// TIA Portal project "sorting task" (V15)

(* hardware
DEVICE "S7300/ET200M station_1"  S7-300 station
   slot 0: "Rail_0"  Rail  6ES7 390-1***0-0AA0
   slot 2: "PLC_1"  CPU 313C-2 DP  6ES7 313-6CF03-0AB0  V2.6
      slot 0: "MPI interface_1"  X1
      slot 1: "DP interface_1"  X2
      slot 2: "DI 16/DO 16_1"  DI16/DO16
      slot 4: "Count_1"  Counter
DEVICE "S7300/ET200M station_2"  S7-300 station
   slot 0: "Rail_0"  Rail  6ES7 390-1***0-0AA0
   slot 2: "PLC_2"  CPU 313C-2 DP  6ES7 313-6CF03-0AB0  V2.6
      slot 0: "MPI interface_1"  X1
      slot 1: "DP interface_1"  X2
      slot 2: "DI 16/DO 16_1"  DI16/DO16
      slot 4: "Count_1"  Counter
*)

// ===== PLC "PLC_1"  CPU 313C-2 DP =====

VAR_GLOBAL   // PLC tag table "Default tag table"
   "Start" AT %I0.5 : Bool;
   "stop" AT %I0.6 : Bool;
   "reset" AT %I0.7 : Bool;
   "L.S" AT %I0.3 : Bool;
   "H.S" AT %I0.4 : Bool;
   "Cyl UP" AT %Q0.0 : Bool;
   "Cyl Down" AT %Q0.1 : Bool;
   "MF" AT %Q0.2 : Bool;
   "MR" AT %Q0.3 : Bool;
   "Suction" AT %Q0.4 : Bool;
   "M1" AT %Q0.5 : Bool;
   "X" AT %M0.0 : Bool;
   "Auto" AT %M41.4 : Bool;
   "Manual" AT %M41.3 : Bool;
   "R1" AT %M0.3 : Bool;
   "R2" AT %M0.4 : Bool;
   "R3" AT %M0.5 : Bool;
   "R4" AT %M0.6 : Bool;
   "R5" AT %M0.7 : Bool;
   "R6" AT %M1.0 : Bool;
   "R7" AT %M1.1 : Bool;
   "R8" AT %M1.2 : Bool;
   "Z1" AT %M2.0 : Bool;
   "Z2" AT %M2.1 : Bool;
   "Z3" AT %M2.2 : Bool;
   "Z4" AT %M2.3 : Bool;
   "Z5" AT %M2.4 : Bool;
   "Z6" AT %M2.5 : Bool;
   "Z7" AT %M2.6 : Bool;
   "Z8" AT %M2.7 : Bool;
   "M11" AT %M32.0 : Bool;
   "M12" AT %M32.1 : Bool;
   "M13" AT %M32.2 : Bool;
   "M14" AT %M32.3 : Bool;
   "M15" AT %M32.4 : Bool;
   "M16" AT %M32.5 : Bool;
   "M17" AT %M32.6 : Bool;
   "M18" AT %M32.7 : Bool;
   "M21" AT %M34.0 : Bool;
   "M22" AT %M34.1 : Bool;
   "M23" AT %M34.2 : Bool;
   "M24" AT %M34.3 : Bool;
   "M25" AT %M34.4 : Bool;
   "M26" AT %M34.5 : Bool;
   "M27" AT %M34.6 : Bool;
   "M28" AT %M34.7 : Bool;
   "P0" AT %M8.0 : Bool;
   "P1" AT %M8.1 : Bool;
   "P2" AT %M8.2 : Bool;
   "P3" AT %M8.3 : Bool;
   "P4" AT %M8.4 : Bool;
   "P5" AT %M8.5 : Bool;
   "P6" AT %M8.6 : Bool;
   "P7" AT %M8.7 : Bool;
   "N0" AT %M9.0 : Bool;
   "N1" AT %M9.1 : Bool;
   "N2" AT %M9.2 : Bool;
   "N3" AT %M9.3 : Bool;
   "N4" AT %M9.4 : Bool;
   "N5" AT %M9.5 : Bool;
   "N6" AT %M9.6 : Bool;
   "N7" AT %M9.7 : Bool;
   "MW20" AT %MW20 : Word;
   "MD100" AT %MD100 : DInt;
   "MD104" AT %MD104 : DInt;
   "C0" AT %M10.0 : Bool;
   "C1" AT %M10.1 : Bool;
   "C2" AT %M10.2 : Bool;
   "C3" AT %M10.3 : Bool;
   "C4" AT %M10.4 : Bool;
   "C5" AT %M10.5 : Bool;
   "C6" AT %M10.6 : Bool;
   "C7" AT %M10.7 : Bool;
   "TON0" AT %M11.0 : Timer;
   "TON1" AT %M11.1 : Bool;
   "TON2" AT %M11.2 : Bool;
   "TON3" AT %M11.3 : Bool;
   "TON4" AT %M11.4 : Bool;
   "TON5" AT %M11.5 : Bool;
   "TON6" AT %M11.6 : Bool;
   "TON7" AT %M11.7 : Bool;
   "T1" AT %M12.0 : Bool;
   "T2" AT %M12.1 : Bool;
   "T3" AT %M12.2 : Bool;
   "T4" AT %M12.3 : Bool;
   "T5" AT %M12.4 : Bool;
   "T6" AT %M12.5 : Bool;
   "T7" AT %M12.6 : Bool;
   "T0" AT %M12.7 : Bool;
   "Large" AT %M13.0 : Bool;
   "small" AT %M13.1 : Bool;
   "B" AT %M13.2 : Bool;
   "u0" AT %M13.3 : Bool;
   "u1" AT %M13.4 : Bool;
   "u2" AT %M13.5 : Bool;
   "u3" AT %M13.6 : Bool;
   "u4" AT %M13.7 : Bool;
   "u5" AT %M14.0 : Bool;
   "u6" AT %M14.1 : Bool;
   "u7" AT %M14.2 : Bool;
   "u8" AT %M14.3 : Bool;
   "u9" AT %M14.4 : Bool;
   "u10" AT %M14.5 : Bool;
   "u11" AT %M14.6 : Bool;
   "u12" AT %M14.7 : Bool;
   "mw88" AT %MW88 : Word;
   "MW30" AT %MW30 : Word;
   "MW32" AT %MW32 : Word;
   "MW34" AT %MW34 : Word;
   "Y" AT %M4.0 : Bool;
   "Y1" AT %M4.1 : Bool;
   "Y2" AT %M4.2 : Bool;
   "Y3" AT %M4.3 : Bool;
   "smll" AT %M4.4 : Bool;
   "up" AT %M40.0 : Bool;
   "down" AT %M40.1 : Bool;
   "left" AT %M40.2 : Bool;
   "right" AT %M40.3 : Bool;
   "suc" AT %M40.4 : Bool;
   "forword" AT %M40.5 : Bool;
   "qw50" AT %QW50 : Word;
   "qw52" AT %QW52 : Word;
   "qw54" AT %QW54 : Word;
   "iw50" AT %IW50 : Word;
   "iw52" AT %IW52 : Word;
   "iw0" AT %IW0 : Word;
   "mw40" AT %MW40 : Word;
   "qw0" AT %QW0 : Word;
   "staart" AT %M41.0 : Bool;
   "stoop" AT %M41.1 : Bool;
   "rese" AT %M41.2 : Bool;
END_VAR

DATA_BLOCK "0"   // DB1
{ S7_Optimized_Access := 'FALSE' }
VERSION : 0.1
// stored: InstanceOfName Negative Age
"Negative Age"
BEGIN
END_DATA_BLOCK

DATA_BLOCK "2"   // DB2
{ S7_Optimized_Access := 'FALSE' }
VERSION : 0.1
// stored: InstanceOfName Negative Age
"Negative Age"
BEGIN
END_DATA_BLOCK

DATA_BLOCK "3"   // DB3
{ S7_Optimized_Access := 'FALSE' }
VERSION : 0.1
// stored: InstanceOfName positive age
"positive age"
BEGIN
END_DATA_BLOCK

DATA_BLOCK "6"   // DB4
{ S7_Optimized_Access := 'FALSE' }
VERSION : 0.1
// stored: InstanceOfName Negative Age
"Negative Age"
BEGIN
END_DATA_BLOCK

DATA_BLOCK "4"   // DB5
{ S7_Optimized_Access := 'FALSE' }
VERSION : 0.1
// stored: InstanceOfName Negative Age
"Negative Age"
BEGIN
END_DATA_BLOCK

DATA_BLOCK "5"   // DB6
{ S7_Optimized_Access := 'FALSE' }
VERSION : 0.1
// stored: InstanceOfName positive age
"positive age"
BEGIN
END_DATA_BLOCK

DATA_BLOCK "7"   // DB7
{ S7_Optimized_Access := 'FALSE' }
VERSION : 0.1
// stored: InstanceOfName positive age
"positive age"
BEGIN
END_DATA_BLOCK

DATA_BLOCK "fb small r8"   // DB8
{ S7_Optimized_Access := 'FALSE' }
VERSION : 0.1
// stored: InstanceOfName FB.SMALL
"FB.SMALL"
BEGIN
END_DATA_BLOCK

DATA_BLOCK "FB.LARGE_R1"   // DB9
{ S7_Optimized_Access := 'FALSE' }
VERSION : 0.1
// stored: InstanceOfName FB.LARGE
"FB.LARGE"
BEGIN
END_DATA_BLOCK

DATA_BLOCK "FB.SMALL_r7"   // DB10
{ S7_Optimized_Access := 'FALSE' }
VERSION : 0.1
// stored: InstanceOfName FB.SMALL
"FB.SMALL"
BEGIN
END_DATA_BLOCK

DATA_BLOCK "FB.SMALL_R6"   // DB11
{ S7_Optimized_Access := 'FALSE' }
VERSION : 0.1
// stored: InstanceOfName FB.SMALL
"FB.SMALL"
BEGIN
END_DATA_BLOCK

DATA_BLOCK "FB.SMALL_R5"   // DB12
{ S7_Optimized_Access := 'FALSE' }
VERSION : 0.1
// stored: InstanceOfName FB.SMALL
"FB.SMALL"
BEGIN
END_DATA_BLOCK

DATA_BLOCK "FB.SMALL_R4"   // DB13
{ S7_Optimized_Access := 'FALSE' }
VERSION : 0.1
// stored: InstanceOfName FB.SMALL
"FB.SMALL"
BEGIN
END_DATA_BLOCK

DATA_BLOCK "FB.SMALL_R3"   // DB14
{ S7_Optimized_Access := 'FALSE' }
VERSION : 0.1
// stored: InstanceOfName FB.SMALL
"FB.SMALL"
BEGIN
END_DATA_BLOCK

DATA_BLOCK "FB.SMALL_R2"   // DB15
{ S7_Optimized_Access := 'FALSE' }
VERSION : 0.1
// stored: InstanceOfName FB.SMALL
"FB.SMALL"
BEGIN
END_DATA_BLOCK

DATA_BLOCK "FB.SMALL_R1"   // DB16
{ S7_Optimized_Access := 'FALSE' }
VERSION : 0.1
// stored: InstanceOfName FB.SMALL
"FB.SMALL"
BEGIN
END_DATA_BLOCK

DATA_BLOCK "FB.LARGE_R2"   // DB17
{ S7_Optimized_Access := 'FALSE' }
VERSION : 0.1
// stored: InstanceOfName FB.LARGE
"FB.LARGE"
BEGIN
END_DATA_BLOCK

DATA_BLOCK "FB.LARGE_R3"   // DB18
{ S7_Optimized_Access := 'FALSE' }
VERSION : 0.1
// stored: InstanceOfName FB.LARGE
"FB.LARGE"
BEGIN
END_DATA_BLOCK

DATA_BLOCK "FB.LARGE_R4"   // DB19
{ S7_Optimized_Access := 'FALSE' }
VERSION : 0.1
// stored: InstanceOfName FB.LARGE
"FB.LARGE"
BEGIN
END_DATA_BLOCK

DATA_BLOCK "FB.LARGE_R5"   // DB20
{ S7_Optimized_Access := 'FALSE' }
VERSION : 0.1
// stored: InstanceOfName FB.LARGE
"FB.LARGE"
BEGIN
END_DATA_BLOCK

DATA_BLOCK "FB.LARGE_R6"   // DB21
{ S7_Optimized_Access := 'FALSE' }
VERSION : 0.1
// stored: InstanceOfName FB.LARGE
"FB.LARGE"
BEGIN
END_DATA_BLOCK

DATA_BLOCK "FB.LARGE_R7"   // DB22
{ S7_Optimized_Access := 'FALSE' }
VERSION : 0.1
// stored: InstanceOfName FB.LARGE
"FB.LARGE"
BEGIN
END_DATA_BLOCK

DATA_BLOCK "FB.LARGE_R8"   // DB23
{ S7_Optimized_Access := 'FALSE' }
VERSION : 0.1
// stored: InstanceOfName FB.LARGE
"FB.LARGE"
BEGIN
END_DATA_BLOCK

DATA_BLOCK "FB.R1"   // DB24
{ S7_Optimized_Access := 'FALSE' }
VERSION : 0.1
// stored: InstanceOfName FB.MR
"FB.MR"
BEGIN
END_DATA_BLOCK

DATA_BLOCK "FB.R2"   // DB25
{ S7_Optimized_Access := 'FALSE' }
VERSION : 0.1
// stored: InstanceOfName FB.MR
"FB.MR"
BEGIN
END_DATA_BLOCK

DATA_BLOCK "FB.R3"   // DB26
{ S7_Optimized_Access := 'FALSE' }
VERSION : 0.1
// stored: InstanceOfName FB.MR
"FB.MR"
BEGIN
END_DATA_BLOCK

DATA_BLOCK "FB.R4"   // DB27
{ S7_Optimized_Access := 'FALSE' }
VERSION : 0.1
// stored: InstanceOfName FB.MR
"FB.MR"
BEGIN
END_DATA_BLOCK

DATA_BLOCK "FB.R5"   // DB28
{ S7_Optimized_Access := 'FALSE' }
VERSION : 0.1
// stored: InstanceOfName FB,MF
"FB,MF"
BEGIN
END_DATA_BLOCK

DATA_BLOCK "FB.R6"   // DB29
{ S7_Optimized_Access := 'FALSE' }
VERSION : 0.1
// stored: InstanceOfName FB,MF
"FB,MF"
BEGIN
END_DATA_BLOCK

DATA_BLOCK "FB.R7"   // DB30
{ S7_Optimized_Access := 'FALSE' }
VERSION : 0.1
// stored: InstanceOfName FB,MF
"FB,MF"
BEGIN
END_DATA_BLOCK

DATA_BLOCK "FB.R8"   // DB31
{ S7_Optimized_Access := 'FALSE' }
VERSION : 0.1
// stored: InstanceOfName FB,MF
"FB,MF"
BEGIN
END_DATA_BLOCK

DATA_BLOCK "Negative Age_last"   // DB33
{ S7_Optimized_Access := 'FALSE' }
VERSION : 0.1
// stored: InstanceOfName Negative Age
"Negative Age"
BEGIN
END_DATA_BLOCK

FUNCTION_BLOCK "Negative Age"   // FB1, SCL
{ S7_Optimized_Access := 'FALSE' }
VERSION : 0.1
   VAR_INPUT
      in : Bool;
   END_VAR
   VAR_OUTPUT
      out : Bool;
   END_VAR
   VAR_IN_OUT
      y : Bool;
   END_VAR
BEGIN
   #out := NOT #in AND #y;
   #y := #y;
END_FUNCTION_BLOCK

FUNCTION_BLOCK "positive age"   // FB2, SCL
{ S7_Optimized_Access := 'FALSE' }
VERSION : 0.1
   VAR_INPUT
      in : Bool;
   END_VAR
   VAR_OUTPUT
      out : Bool;
   END_VAR
   VAR_IN_OUT
      y : Bool;
   END_VAR
BEGIN
   #out := #in AND NOT #y;
   #y := #in;
END_FUNCTION_BLOCK

FUNCTION_BLOCK "Block_1"   // FB3, LAD
{ S7_Optimized_Access := 'FALSE' }
VERSION : 0.1
   VAR_TEMP   // added for the SCL form of the ladder/FBD networks
      _s5time1 : S5Time;
   END_VAR
BEGIN

REGION Network 1
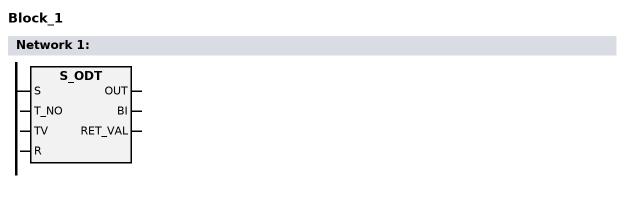
   RUNG wire#powerrail
      S_ODT(T_NO :=, TV :=, R :=, BI =>, RET_VAL =>)
   END_RUNG
   // the same network as SCL:
   #_s5time1 := S_ODT(S := TRUE);
END_REGION
END_FUNCTION_BLOCK

FUNCTION_BLOCK "FB.SMALL"   // FB4, SCL
{ S7_Optimized_Access := 'FALSE' }
VERSION : 0.1
BEGIN
   "R8" := NOT "M18";
   "R7" := NOT "M17" AND NOT "R8";
   "R6" := NOT "M16" AND NOT "R8" AND NOT "R7" ;
   "R5" := NOT "M15" AND NOT "R8" AND NOT "R7" AND NOT "R6" ;
   "R4" := NOT "M14" AND NOT "R8" AND NOT "R7" AND NOT "R6" AND NOT "R5";
   "R3" := NOT "M13" AND NOT "R8" AND NOT "R7" AND NOT "R6" AND NOT "R5" AND NOT "R4" ;
   "R2" := NOT "M12" AND NOT "R8" AND NOT "R7" AND NOT "R6" AND NOT "R5" AND NOT "R4" AND NOT "R3";
   "R1" := NOT "M11" AND NOT "R8" AND NOT "R7" AND NOT "R6" AND NOT "R5" AND NOT "R4" AND NOT "R3" AND NOT "R2";
   IF "R8"=1 AND "Y"=1 THEN
       SET(S_BIT:="M18",N:=1);
   END_IF;
   IF "R7" = 1 AND "Y" = 1 THEN
       SET(S_BIT := "M17",N := 2);
   END_IF;
   IF "R6" = 1 AND "Y" = 1 THEN
       SET(S_BIT := "M16",N := 3);
   END_IF;
   IF "R5" = 1 AND "Y" = 1 THEN
       SET(S_BIT := "M15",N := 4);
   END_IF;
   IF "R4" = 1 AND "Y" = 1 THEN
       SET(S_BIT := "M14",N := 5);
   END_IF;
   IF "R3" = 1 AND "Y" = 1 THEN
       SET(S_BIT := "M13", N := 6);
   END_IF;
   IF "R2" = 1 AND "Y" = 1 THEN
       SET(S_BIT := "M12", N := 7);
   END_IF;
   IF "R1" = 1 AND "Y" = 1 THEN
       SET(S_BIT := "M11", N := 8);
   END_IF;
END_FUNCTION_BLOCK

FUNCTION_BLOCK "FB.LARGE"   // FB5, SCL
{ S7_Optimized_Access := 'FALSE' }
VERSION : 0.1
BEGIN
   "R1" := "M21";
   "R2" := "M22" AND NOT "R1";
   "R3" := "M23" AND NOT "R1" AND NOT "R2";
   "R4" := "M24" AND NOT "R1" AND NOT "R2" AND NOT "R3";
   "R5" := "M25" AND NOT "R1" AND NOT "R2" AND NOT "R3" AND NOT "R4";
   "R6" := "M26" AND NOT "R1" AND NOT "R2" AND NOT "R3" AND NOT "R4" AND NOT "R5";
   "R7" := "M27" AND NOT "R1" AND NOT "R2" AND NOT "R3" AND NOT "R4" AND NOT "R5" AND NOT "R6";
   "R8" := "M28" AND NOT "R1" AND NOT "R2" AND NOT "R3" AND NOT "R4" AND NOT "R5" AND NOT "R6" AND NOT "R7";
   IF "R1"=1 AND "Y"=1THEN
       RESET(S_BIT:="M21", N:=1);
   END_IF;
   IF "R2" = 1 AND "Y" = 1 THEN
       RESET(S_BIT := "M22",
             N := 2);
   END_IF;
   IF "R3" = 1 AND "Y" = 1 THEN
       RESET(S_BIT := "M23",
             N := 3);
   END_IF;
   IF "R4" = 1 AND "Y" = 1 THEN
       RESET(S_BIT := "M24",
             N := 4);
   END_IF;
   IF "R5" = 1 AND "Y" = 1 THEN
       RESET(S_BIT := "M25",
             N := 5);
   END_IF;
   IF "R6" = 1 AND "Y" = 1 THEN
       RESET(S_BIT := "M26",
             N := 6);
   END_IF;
   IF "R7" = 1 AND "Y" = 1 THEN
       RESET(S_BIT := "M27",
             N := 7);
   END_IF;
   IF "R8" = 1 AND "Y" = 1 THEN
       RESET(S_BIT := "M28",
             N := 8);
   END_IF;
END_FUNCTION_BLOCK

FUNCTION_BLOCK "FB.MR"   // FB6, SCL
{ S7_Optimized_Access := 'FALSE' }
VERSION : 0.1
   VAR_INPUT
      MD110 : DInt;
   END_VAR
   VAR
      P00 : Bool;
      T00 : Bool;
      T11 : Bool;
      T22 : Bool;
      T33 : Bool;
      T44 : Bool;
      T55 : Bool;
      T66 : Bool;
      T77 : Bool;
      T88 : Bool;
      MW88 : Word;
      U00 : Bool;
      U11 : Bool;
      U22 : Bool;
      U33 : Bool;
   END_VAR
BEGIN
   "7"(in:="T1",out=>#P00, y:=#U00);
   IF #P00=1 THEN
       SET(S_BIT:="Cyl Down",  N:=9);
   END_IF;

   #MW88:= S_ODT(T_NO:=10, S:="Cyl Down"AND NOT "Suction", TV:=S5T#500MS, Q=>#T11);
   IF #T11=1 THEN
       RESET(S_BIT:="Cyl Down",
             N:=10);
       SET(S_BIT:="Suction",
           N:=11);
       SET(S_BIT:="Cyl UP",
           N:=12);
   END_IF;

   #MW88 := S_ODT(T_NO := 11, S := "Cyl UP" AND "Suction", TV := S5T#500MS, Q => #T22);
   IF #T22 = 1 THEN
       RESET(S_BIT := "Cyl UP",
             N := 13);
       SET(S_BIT := "MR",
           N := 14);
       SET(S_BIT := "Y",
           N := 15);
   END_IF;
   IF "MD100" < #MD110 AND "Suction" = 1 THEN
       RESET(S_BIT := "MR",
             N := 16);
   END_IF;
   IF "R1" = 1 AND "Suction" = 1 AND "MR" = 0 THEN
       SET(S_BIT := "Cyl Down",
           N := 17);
   END_IF;
   #MW88 := S_ODT(T_NO := 12, S := "Cyl Down" AND "Suction", TV := S5T#500MS, Q => #T33);
   IF #T33 = 1 THEN
       RESET(S_BIT := "Cyl Down",
             N := 18);
       RESET(S_BIT := "Suction",
             N := 19);
       SET(S_BIT := "Cyl UP",
           N := 20);
   END_IF;
   #MW88 := S_ODT(T_NO := 13, S := "Cyl UP" AND NOT "Suction", TV := S5T#500MS, Q => #T44);
   IF #T44 = 1 THEN
       RESET(S_BIT := "Cyl UP",
             N := 21);
       RESET(S_BIT := "Y",
             N := 22);
   END_IF;
END_FUNCTION_BLOCK

FUNCTION_BLOCK "FB,MF"   // FB7, SCL
{ S7_Optimized_Access := 'FALSE' }
VERSION : 0.1
   VAR_INPUT
      MD110 : DInt;
   END_VAR
   VAR
      P00 : Bool;
      T00 : Bool;
      T11 : Bool;
      T22 : Bool;
      T33 : Bool;
      T44 : Bool;
      T55 : Bool;
      T66 : Bool;
      T77 : Bool;
      T88 : Bool;
      MW88 : Word;
      U00 : Bool;
      U11 : Bool;
      U22 : Bool;
      U33 : Bool;
   END_VAR
BEGIN
   "7"(in := "T1",
       out => #P00,
       y := #U00);
   IF #P00 = 1 THEN
       SET(S_BIT := "Cyl Down",
           N := 9);
   END_IF;

   #MW88 := S_ODT(T_NO := 10, S := "Cyl Down" AND NOT "Suction", TV := S5T#500MS, Q => #T11);
   IF #T11 = 1 THEN
       RESET(S_BIT := "Cyl Down",
             N := 10);
       SET(S_BIT := "Suction",
           N := 11);
       SET(S_BIT := "Cyl UP",
           N := 12);
   END_IF;

   #MW88 := S_ODT(T_NO := 11, S := "Cyl UP" AND "Suction", TV := S5T#500MS, Q => #T22);
   IF #T22 = 1 THEN
       RESET(S_BIT := "Cyl UP",
             N := 13);
       SET(S_BIT := "MF",
           N := 14);
       SET(S_BIT := "Y",
           N := 15);
   END_IF;
   IF "MD100" > #MD110 AND "Suction" = 1 THEN
       RESET(S_BIT := "MF",
             N := 16);
   END_IF;
   IF "R1" = 1 AND "Suction" = 1 AND "MR" = 0 THEN
       SET(S_BIT := "Cyl Down",
           N := 17);
   END_IF;
   #MW88 := S_ODT(T_NO := 12, S := "Cyl Down" AND "Suction", TV := S5T#500MS, Q => #T33);
   IF #T33 = 1 THEN
       RESET(S_BIT := "Cyl Down",
             N := 18);
       RESET(S_BIT := "Suction",
             N := 19);
       SET(S_BIT := "Cyl UP",
           N := 20);
   END_IF;
   #MW88 := S_ODT(T_NO := 13, S := "Cyl UP" AND NOT "Suction", TV := S5T#500MS, Q => #T44);
   IF #T44 = 1 THEN
       RESET(S_BIT := "Cyl UP",
             N := 21);
       RESET(S_BIT:="Y",
             N:=22);

   END_IF;
END_FUNCTION_BLOCK

ORGANIZATION_BLOCK "Main"   // OB1, SCL
TITLE = "Main Program Sweep (Cycle)"
{ S7_Optimized_Access := 'FALSE' }
VERSION : 0.1
   VAR_TEMP
      OB1_EV_CLASS : Byte;   // Bits 0-3 = 1 (Coming event), Bits 4-7 = 1 (Event class 1)
      OB1_SCAN_1 : Byte;   // 1 (Cold restart scan 1 of OB 1), 3 (Scan 2-n of OB 1)
      OB1_PRIORITY : Byte;   // Priority of OB Execution
      OB1_OB_NUMBR : Byte;   // 1 (Organization block 1, OB1)
      OB1_RESERVED_1 : Byte;   // Reserved for system
      OB1_RESERVED_2 : Byte;   // Reserved for system
      OB1_PREV_CYCLE : Int;   // Cycle time of previous OB1 scan (milliseconds)
      OB1_MIN_CYCLE : Int;   // Minimum cycle time of OB1 (milliseconds)
      OB1_MAX_CYCLE : Int;   // Maximum cycle time of OB1 (milliseconds)
      OB1_DATE_TIME : Date_And_Time;   // Date and time OB1 started
   END_VAR
BEGIN
   REGION "X"
       "X" := ("Start" OR "X" OR "staart") AND "stop" AND "stoop" AND "Auto";
       "5"(in:="X",out=>"P1", y:="u4");
       IF "P1"=1 AND "X"=1  THEN
           "MW32" := "MW30";
           "MW34" := "MW30";
           SET(S_BIT:= "Y1",
               N:=50);

       END_IF;


   END_REGION

   REGION encoder
       "encoder"(LADDR:=16#300,
                 CHANNEL:=0,
                 SW_GATE:="Y1",
                 COUNTVAL=>"MD100");

              END_REGION


   IF "MD100"<5 AND "MD100">-5 THEN
       "M1":="X" AND NOT "Suction";
   ELSE
       "M1" := 0;
   END_IF;

   "0"(in:="H.S", out=>"Large", y:="N0");
   "2"(in:="L.S",out=>"N1", y:="u0");
   "small" := "N1" AND NOT "H.S" AND NOT "Large";

   IF "MD100"<5 AND "MD100">-5 THEN
       "3"(in:=TRUE, out=>"P0", y:="u1");
       IF "MD100"<5 AND "MD100">-5 AND "P0"=1 THEN
           RESET(S_BIT:="Large",
                 N:=32);
           RESET(S_BIT:="small",
                 N:=33);
           RESET(S_BIT:="smll",
                 N:=34);
           RESET(S_BIT := "B",
                 N := 35);
       END_IF;
   END_IF;

   "6"(in:="L.S",out=>"N2", y:="u2");
   "mw88" := S_CU(C_NO := 106, CU := "N2", R:="u8", CV=>"MW20");

   REGION RePosition
       "4"(in := "Suction",
      out => "N3",
      y := "u3");
       IF "N3" = 1 THEN
           SET(S_BIT := "B",
          N := 40);
       END_IF;
       "mw88" := S_ODT(T_NO := 1, S := "B", TV := s5t#600ms, Q => "T2");
       (*
       لو فيه مشكله ان الماتور لما ييجي يرجع للنص 
       ومش بيقف ساعتها اعمل ايلسي لل الكود اللي جاي
       *)
       IF "MD100" < -5 AND "T2" = 1 THEN
           "MF" := 1;

       END_IF;
       IF "MD100" > 5 AND "T2" = 1 THEN
           "MR" := 1;
       END_IF;
   END_REGION


   (*
   التايمر اللي تحت ده الوقت بتاعه هبتغير علي حسب الوقت اللي هيقف فيه السير
   *)
   IF "N1" = 1 THEN
       SET(S_BIT := "smll",
           N := 31);
   END_IF;


   "mw88" := S_ODT(T_NO := 3, S := "smll", TV := S5T#1.5S, Q=>"T1");
   IF "T1" = 1 THEN
       RESET(S_BIT := "M1",
             N := 30);
   END_IF;

   REGION small

   IF "T1" = 1 AND "small" = 1 AND "MW20" = 1 THEN
       "fb small r8"();
   END_IF;
   IF "T1" = 1 AND "small" = 1 AND "MW20" = 2 THEN
       "FB.SMALL_r7"();
   END_IF;
   IF "T1" = 1 AND "small" = 1 AND "MW20" = 3 THEN
       "FB.SMALL_R6"();
   END_IF;
   IF "T1" = 1 AND "small" = 1 AND "MW20" = 4 THEN
       "FB.SMALL_R5"();
   END_IF;
   IF "T1" = 1 AND "small" = 1 AND "MW20" = 5 THEN
       "FB.SMALL_R4"();
   END_IF;
   IF "T1" = 1 AND "small" = 1 AND "MW20" = 6 THEN
       "FB.SMALL_R3"();
   END_IF;
   IF "T1" = 1 AND "small" = 1 AND "MW20" = 7 THEN
       "FB.SMALL_R2"();
   END_IF;
   IF "T1" = 1 AND "small" = 1 AND "MW20" = 8 THEN
       "FB.SMALL_R1"();
   END_IF;

   END_REGION

   REGION large
       IF "Large" = 1 AND "T1" = 1 AND "MW20" = 1 THEN
           "FB.LARGE_R1"();
       END_IF;
       IF "Large" = 1 AND "T1" = 1 AND "MW20" = 2 THEN
           "FB.LARGE_R2"();
       END_IF;
       IF "Large" = 1 AND "T1" = 1 AND "MW20" = 2 THEN
           "FB.LARGE_R3"();
       END_IF;
       IF "Large" = 1 AND "T1" = 1 AND "MW20" = 2 THEN
           "FB.LARGE_R4"();
       END_IF;
       IF "Large" = 1 AND "T1" = 1 AND "MW20" = 2 THEN
           "FB.LARGE_R5"();
       END_IF;
       IF "Large" = 1 AND "T1" = 1 AND "MW20" = 2 THEN
           "FB.LARGE_R6"();
       END_IF;
       IF "Large" = 1 AND "T1" = 1 AND "MW20" = 2 THEN
           "FB.LARGE_R7"();
       END_IF;
       IF "Large" = 1 AND "T1" = 1 AND "MW20" = 2 THEN
           "FB.LARGE_R8"();
       END_IF;

   END_REGION

   REGION POSITION R1
       IF "R1" = 1 THEN
           "FB.R1"(-500);
       END_IF;
   END_REGION

   REGION POSITION R2
       IF "R2" = 1 THEN
           "FB.R2"(-400);
       END_IF;
   END_REGION

   REGION POSITION R3
       IF "R3" = 1 THEN
           "FB.R3"(-300);
       END_IF;
   END_REGION

   REGION POSITION R4
       IF "R4" = 1 THEN
           "FB.R4"(-200);
       END_IF;
   END_REGION

   REGION POSITION R5
       IF "R5" = 1 THEN
           "FB.R5"(200);
       END_IF;
   END_REGION

   REGION POSITION R6
       IF "R6" =1 THEN
      "FB.R6"(300);
       END_IF;
   END_REGION

   REGION POSITION R7
       IF "R7" = 1 THEN
           "FB.R7"(400);
       END_IF;
   END_REGION

   REGION POSITION R8
       IF "R8" = 1 THEN
           "FB.R8"(500);
       END_IF;
   END_REGION

   REGION close program
       "Negative Age_last"(in:="B", out=>"N5",y:="u7");
       IF "N5" = 1 AND "MW20" = 8 THEN
           RESET(S_BIT:="X",
                 N:=41);
           "u8" := 1;

       END_IF;

   END_REGION

   REGION reset
       IF "reset" = 1 OR "rese"=1 THEN
           SET(S_BIT := "Y2",
               N := 51);
       END_IF;
       IF "Y2" = 1 THEN
           IF "MD100" > 5 THEN
               "MR" := 1;
           ELSE
               "MR" := 0;
           END_IF;
           IF "MD100" < -5 THEN
               "MF" := 1;
           ELSE
               "MF" := 0;
           END_IF;
           IF "MD100"<10 AND "MD100">-10 THEN
               RESET(S_BIT := "Y2",
                     N := 45);
           END_IF;

       END_IF;
   END_REGION

   REGION manual
       IF "Manual"=1 AND "Auto" =0 THEN
           "Cyl Down" := "down";
           "Cyl UP" := "up";
           "MF" := "left";
           "MR" := "right";
           "Suction" := "suc";
           "M1" := "forword";
       END_IF;

   END_REGION

   REGION communication
       "qw50" := "iw0";
       "qw52" := "qw0"; 
       "mw40" := "iw50";
       "MW30" := "iw52";
       "qw54" := "MW30";



   END_REGION
END_ORGANIZATION_BLOCK

// ===== PLC "PLC_2"  CPU 313C-2 DP =====

VAR_GLOBAL   // PLC tag table "Default tag table"
   "mw0" AT %MW0 : Word;
   "iw50" AT %IW50 : Word;
   "iw52" AT %IW52 : Word;
   "iw54" AT %IW54 : Word;
   "qw50" AT %QW50 : Word;
   "qw52" AT %QW52 : Word;
   "mw10" AT %QW54 : Word;
   "mw40" AT %QW56 : Word;
   "mw30" AT %QW58 : Word;
END_VAR

ORGANIZATION_BLOCK "Main"   // OB1, SCL
TITLE = "Main Program Sweep (Cycle)"
{ S7_Optimized_Access := 'FALSE' }
VERSION : 0.1
   VAR_TEMP
      OB1_EV_CLASS : Byte;   // Bits 0-3 = 1 (Coming event), Bits 4-7 = 1 (Event class 1)
      OB1_SCAN_1 : Byte;   // 1 (Cold restart scan 1 of OB 1), 3 (Scan 2-n of OB 1)
      OB1_PRIORITY : Byte;   // Priority of OB Execution
      OB1_OB_NUMBR : Byte;   // 1 (Organization block 1, OB1)
      OB1_RESERVED_1 : Byte;   // Reserved for system
      OB1_RESERVED_2 : Byte;   // Reserved for system
      OB1_PREV_CYCLE : Int;   // Cycle time of previous OB1 scan (milliseconds)
      OB1_MIN_CYCLE : Int;   // Minimum cycle time of OB1 (milliseconds)
      OB1_MAX_CYCLE : Int;   // Maximum cycle time of OB1 (milliseconds)
      OB1_DATE_TIME : Date_And_Time;   // Date and time OB1 started
   END_VAR
BEGIN
   "mw0" := "iw50";
   "mw10" := "iw52";
   "qw50" := "mw40";
   "mw30" := "iw54";
   "qw52" := "mw30";
END_ORGANIZATION_BLOCK